// TIA Portal V20 export
TYPE "type_emRelations_em12_cmStatus"
// stored: Access Published, Namespace Unit1
   STRUCT
      StackNgBoxDetect : "LBC_typeDigitalSignalControlNode";
      StackNgBoxFullDetect : "LBC_typeDigitalSignalControlNode";
      StackNgBoxLoadingUpDown : "LBC_typeTwoWayActuatorControlNode";
      StackNgBoxUnitMoverBwdFwd : "LBC_typeTwoWayActuatorControlNode";
      StackNgBoxClampLeftOpenClose : "LBC_typeTwoWayActuatorControlNode";
      StackNgBoxClampRightOpenClose : "LBC_typeTwoWayActuatorControlNode";
      StackNgBoxClampMoverOpenClose : "LBC_typeTwoWayActuatorControlNode";
      StackNgBoxLiftDownUp : "LBC_typeTwoWayActuatorControlNode";
      StackNgBoxLockDownUp : "LBC_typeTwoWayActuatorControlNode";
   END_STRUCT;
END_TYPE
